TYPE Out_16_To_PLC :
STRUCT
	Out AT %I*:ARRAY [1..16] OF BOOL;
END_STRUCT
END_TYPE

(* stored: Version 1.1.0.1, ProductVersion 3.1.4024.15
   DUT Out_16_To_PLC: Id {a6a26fd0-ca0f-4305-8ef4-011bde3ff595} *)
